TYPE ConfigManagerStatuses :
STRUCT
	///Is the config manager in a busy state?
	busyStatus: BusyStatus;
	///Is the config manager in a healthy state?
	healthStatus: HealthStatus;
END_STRUCT
END_TYPE

(* stored: Version 1.1.0.1, ProductVersion 3.1.4019.2
   DUT ConfigManagerStatuses: Id {3f87d15c-8e82-45c4-aba0-8ed0e09f72c2} *)
